FOR i := 0 TO _config.MaxControledUnits DO
    IF _controlledUnits[i] <> 0 THEN
        _status.State.AllInAuto := _status.State.AllInAuto AND _controlledUnits[i].StatusInfo.Mode = eCUMode.AutomatMode;
        _status.State.AllInManual := _status.State.AllInManual AND _controlledUnits[i].StatusInfo.Mode = eCUMode.ManualMode;
        _status.State.AllIdle := _status.State.AllIdle AND _controlledUnits[i].StatusInfo.Mode = eCUMode.NoMode;
        _status.State.AllInGrounding := _status.State.AllInGrounding AND
            (_controlledUnits[i].StatusInfo.Mode = eCUMode.GroundModeDone XOR
            _controlledUnits[i].StatusInfo.Mode = eCUMode.GroundMode);
        _status.State.AllGrounded := _status.State.AllGrounded AND _controlledUnits[i].StatusInfo.Mode = eCUMode.GroundModeDone;
        _status.State.AllInStepMode := _status.State.AllInStepMode AND _controlledUnits[i].StatusInfo.CurrentIsInStepMode;
        _status.State.AllSuspended := _status.State.AllSuspended AND _controlledUnits[i].SuspendTask.Task.Done;
		_status.State.AllRecovered := _status.State.AllRecovered AND _controlledUnits[i].RecoverTask.Task.Done;
		_status.State.AllInactiveOrManualOrGrounded := _status.State.AllInactiveOrManualOrGrounded 
											AND (_controlledUnits[i].StatusInfo.Mode = eCUMode.ManualMode 
												OR _controlledUnits[i].StatusInfo.Mode = eCUMode.NoMode 
												OR _controlledUnits[i].StatusInfo.Mode = eCUMode.GroundModeDone );
		
        _status.State.AnyInAuto := _status.State.AnyInAuto OR _controlledUnits[i].StatusInfo.Mode = eCUMode.AutomatMode;
        _status.State.AnyInManual := _status.State.AnyInManual OR _controlledUnits[i].StatusInfo.Mode = eCUMode.ManualMode;
        _status.State.AnyInStepMode := _status.State.AnyInStepMode OR _controlledUnits[i].StatusInfo.CurrentIsInStepMode;
        _status.State.AnyGrounding := _status.State.AnyGrounding OR
            (_controlledUnits[i].StatusInfo.Mode = eCUMode.GroundModeDone OR
            _controlledUnits[i].StatusInfo.Mode = eCUMode.GroundMode);

    ELSE
        EXIT;
    END_IF
END_FOR

// update states of buttons
_status.State.AnyButtonRecover := FALSE;
_status.State.AnyButtonSuspend := FALSE;
_status.State.AnyButtonGround := FALSE;
_status.State.AnyButtonAuto := FALSE;
i := 0;

FOR i := 0 TO _config.MaxControlButtons DO
    IF _controlButtons[i] <> 0 THEN
        _status.State.AnyButtonRecover := _status.State.AnyButtonRecover OR _controlButtons[i].ButtonRecover;
        _status.State.AnyButtonGround := _status.State.AnyButtonGround OR _controlButtons[i].ButtonGround;
        _status.State.AnyButtonAuto := _status.State.AnyButtonAuto OR _controlButtons[i].ButtonAuto;
        _status.State.AnyButtonSuspend := _status.State.AnyButtonSuspend OR _controlButtons[i].ButtonSuspend;
    ELSE
        EXIT;
    END_IF
END_FOR

// update states of keys
_status.State.AllKeysNormal := TRUE;
_status.State.AnyKeyService := FALSE;
i := 0;

FOR i := 0 TO _config.MaxKeyNormalService DO
    IF _controlKeyNormalService[i] <> 0 THEN
        _status.State.AllKeysNormal := _status.State.AllKeysNormal AND _controlKeyNormalService[i].KeyInNormal;
        _status.State.AnyKeyService := _status.State.AnyKeyService OR _controlKeyNormalService[i].KeyInService;
    ELSE
        EXIT;
    END_IF
END_FOR

// update states of keys
_status.State.AllKeysAuto := TRUE;
_status.State.AnyKeyManual := FALSE;
_status.State.AnyKeyStep := FALSE;
i := 0;

FOR i := 0 TO _config.MaxKeyMode DO
    IF _controlKeyMode[i] <> 0 THEN
        _status.State.AllKeysAuto := _status.State.AllKeysAuto AND _controlKeyMode[i].KeyInAuto;
        _status.State.AnyKeyManual := _status.State.AnyKeyManual OR _controlKeyMode[i].KeyInManual;
        _status.State.AnyKeyStep := _status.State.AnyKeyStep OR _controlKeyMode[i].KeyInStep;
    ELSE
        EXIT;
    END_IF
END_FOR
END_METHOD

METHOD KeyAuto 
VAR
	cu : UINT;
END_VAR
IF _keyAutoTask.Execute() THEN
	_status.ActionDescription:= '<#Automatic mode is not possibe to set(All keys must be in NORMAL and AUTO!)#>';
	IF 	 _status.State.AllKeysNormal  AND _status.State.AllKeysAuto THEN
		
//			_status.ActionDescription:= '<#Automatic mode is set(Step mode is disabled)!#>';
//			FOR cu := 0 TO _config.MaxControledUnits DO
//				IF _controlledUnits[cu] <> 0 THEN
//					IF _controlledUnits[cu].StatusInfo.Mode=eCUMode.AutomatMode THEN
//						_controlledUnits[cu].AutomatTask.ModeController.Mode:=eSequencerMode.CyclicMode;
//					ELSIF _controlledUnits[cu].StatusInfo.Mode=eCUMode.GroundMode THEN
//						_controlledUnits[cu].GroundTask.ModeController.Mode:=eSequencerMode.CyclicMode;
//					END_IF
//				ELSE
//					EXIT;
//				END_IF
//			END_FOR
	
		ELSE
			_status.ActionDescription:= '<#Cyclic mode is not allowed while any control key is in Service mode!#> <#Setting step mode!#>';
			FOR cu := 0 TO _config.MaxControledUnits DO
				IF _controlledUnits[cu] <> 0 THEN
						IF _controlledUnits[cu].StatusInfo.Mode=eCUMode.AutomatMode THEN
							_controlledUnits[cu].AutomatTask.ModeController.Mode:=eSequencerMode.StepMode;
						ELSIF _controlledUnits[cu].StatusInfo.Mode=eCUMode.GroundMode THEN
							_controlledUnits[cu].GroundTask.ModeController.Mode:=eSequencerMode.StepMode;
						END_IF
				ELSE
					EXIT;
				END_IF
			END_FOR	
		END_IF;
	
	


	IF  _status.State.AllInAuto THEN
		_keyAutoTask.DoneWhen(TRUE);
	END_IF;
	
	IF _status.ActionDescription<>'' THEN
		THIS^._keyAutoTask.Messenger.Notify(_status.ActionDescription);
	END_IF;	
END_IF
END_METHOD

METHOD KeyManual 
VAR
	cu : UINT;
END_VAR

IF _keyManualTask.Execute() THEN
	_status.ActionDescription:= '<#Manual mode is not possibe to set(At least one SERVICE and one MANUAL keys must be in position!)#>';
	
	IF _keyManualTask.Progress =0 THEN
		IF _status.State.AnyKeyManual AND _status.State.AnyKeyService THEN
			IF NOT _status.State.AllInManual THEN
				_keyManualTask.Progress := _keyManualTask.Progress + 1;// all to manual
			ELSE
				_keyManualTask.Progress := _keyManualTask.Progress + 2;
			END_IF
		END_IF;
	
	END_IF

	IF _keyManualTask.Progress =1 THEN
		
		_status.ActionDescription:='<#Manual mode is starting#>';
		
		FOR cu := 0 TO _config.MaxControledUnits DO
			IF _controlledUnits[cu] <> 0 THEN
				IF  _controlledUnits[cu].StatusInfo.Mode<> eCUMode.ManualMode THEN
					_controlledUnits[cu].ManualTask.Invoke();
				END_IF			
			ELSE
				EXIT;
			END_IF
		END_FOR

		IF _status.State.AllInManual THEN
			_keyManualTask.Progress := _keyManualTask.Progress + 1;
		END_IF
		
	END_IF
	
	
	IF _keyManualTask.Progress =2 THEN
		
		_status.ActionDescription:='<#Clear step mode#>';
		
		FOR cu := 0 TO _config.MaxControledUnits DO
			IF _controlledUnits[cu] <> 0 THEN
				_controlledUnits[cu].AutomatTask.ModeController.Mode := eSequencerMode.CyclicMode;
				_controlledUnits[cu].GroundTask.ModeController.Mode := eSequencerMode.CyclicMode;		
			ELSE
				EXIT;
			END_IF
		END_FOR

		IF _status.State.AllInManual THEN
			_keyManualTask.Progress := _keyManualTask.Progress + 1;
		END_IF
		
	END_IF

	IF _keyManualTask.Progress =3 THEN
		_keyManualTask.DoneWhen(TRUE);	
	END_IF

	IF _status.ActionDescription<>'' THEN
		THIS^._keyManualTask.Messenger.Notify(_status.ActionDescription);
	END_IF;
END_IF;
END_METHOD

METHOD KeyService
VAR
	cu : UINT;
END_VAR
IF _keyServiceTask.Execute() THEN
	
	IF 	_status.State.AnyKeyManual  AND _status.State.AnyKeyService  THEN
		_status.ActionDescription:='<#Manual mode is starting due service key combination (Manual / Service)#>';
		
		FOR cu := 0 TO _config.MaxControledUnits DO
			IF _controlledUnits[cu] <> 0 THEN
				IF  _controlledUnits[cu].StatusInfo.Mode<> eCUMode.ManualMode THEN
					_controlledUnits[cu].ManualTask.Invoke();
				END_IF			
			ELSE
				EXIT;
			END_IF
		END_FOR
	ELSE
		_status.ActionDescription:='<#Step mode is required because Service key position is set!#>';
		FOR cu := 0 TO _config.MaxControledUnits DO
			IF _controlledUnits[cu] <> 0 THEN
					IF _controlledUnits[cu].StatusInfo.Mode=eCUMode.AutomatMode THEN
						_controlledUnits[cu].AutomatTask.ModeController.Mode:=eSequencerMode.StepMode;
					ELSIF _controlledUnits[cu].StatusInfo.Mode=eCUMode.GroundMode THEN
						_controlledUnits[cu].GroundTask.ModeController.Mode:=eSequencerMode.StepMode;
					END_IF
			ELSE
				EXIT;
			END_IF
		END_FOR
	END_IF;
	


	IF  _status.State.AllInStepMode OR _status.State.AllInManual THEN
		_keyServiceTask.DoneWhen(TRUE);
	END_IF;
	
	IF _status.ActionDescription<>'' THEN
		THIS^._keyServiceTask.Messenger.Notify(_status.ActionDescription);
	END_IF;	
END_IF
END_METHOD

METHOD KeyStep 
VAR
	cu : UINT;
END_VAR

IF _keyStepTask.Execute() THEN
		
	_status.ActionDescription:='<#Step mode is required but mode key is not in required position!#>';

	IF _status.State.AnyKeyStep THEN
		FOR cu := 0 TO _config.MaxControledUnits DO
			IF _controlledUnits[cu] <> 0 THEN
				IF _controlledUnits[cu].StatusInfo.Mode=eCUMode.AutomatMode THEN
					_controlledUnits[cu].AutomatTask.ModeController.Mode:=eSequencerMode.StepMode;
				ELSIF _controlledUnits[cu].StatusInfo.Mode=eCUMode.GroundMode THEN
					_controlledUnits[cu].GroundTask.ModeController.Mode:=eSequencerMode.StepMode;
				END_IF
			ELSE
				EXIT;
			END_IF
		
		END_FOR
	END_IF;
	
	IF _status.State.AllInStepMode THEN
		_status.ActionDescription:='<#Step mode is set or all are inactive!#>';
		_keyStepTask.DoneWhen(TRUE);
	END_IF;
	
	IF _status.ActionDescription<>'' THEN
		THIS^._keyStepTask.Messenger.Notify(_status.ActionDescription);
	END_IF;	
END_IF;
END_METHOD

METHOD Restore :  TcoCore.ITcoRestorable
VAR
	i : UINT;
END_VAR
// clear all linked Controlled units
FOR i := 0 TO _config.MaxControledUnits DO
	_controlledUnits[i] := 0;
END_FOR

// clear all linked Control buttons
FOR i := 0 TO _config.MaxControlButtons DO
	_controlButtons[i] := 0;
END_FOR

// clear all linked service keys (N/S)
FOR i := 0 TO _config.MaxKeyNormalService DO
	_controlKeyNormalService[i] := 0;
END_FOR

// clear all linked Sequencer keys (M/S/A)
FOR i := 0 TO _config.MaxKeyMode DO
	_controlKeyMode[i] := 0;
END_FOR


THIS^.Messenger.UnPin();
END_METHOD

(*~
	<docu>
		<summary>
		    Custom service (manual, maintenance) logic.
			This method must be implemented in derived class.
		</summary>			
	</docu>	
~*)
METHOD PROTECTED  ServiceMode
END_METHOD

METHOD Signalisation
VAR_INPUT
END_VAR

AnyButtonAuto:=_blinkerSlow.IsOn  AND _autoTask.Busy;
END_METHOD

PROPERTY Status : REFERENCE TO TcoControlledZone_Status
GET
Status REF=_status;
END_GET
END_PROPERTY

END_FUNCTION_BLOCK

// ---- Abstractions/Safety/ControlVoltage/TcoControlVoltage.TcPOU
{attribute wpf [Container(Layout.Stack)]}
FUNCTION_BLOCK TcoControlVoltage EXTENDS TcoElements.TcoDi IMPLEMENTS  ITcoControlVoltage

VAR_OUTPUT
END_VAR
VAR
END_VAR

SUPER^(inoSignal:=inoSignal);
IF NOT inoSignal THEN
	Messenger.Error('<#Voltage is Off!#>');
END_IF;

PROPERTY IsOff : BOOL
GET
IsOff:=not this^._signal;
END_GET
END_PROPERTY

PROPERTY IsOn : BOOL
GET
IsOn:=this^._signal;
END_GET
END_PROPERTY

END_FUNCTION_BLOCK

// ---- Abstractions/Safety/DoorCircuit/TcoDoorCircuit.TcPOU
FUNCTION_BLOCK TcoDoorCircuit EXTENDS TcoCore.TcoComponent IMPLEMENTS ITcoDoorCircuit
VAR_INPUT
END_VAR
VAR_OUTPUT
END_VAR
VAR
	
	{attribute addProperty Name "<#Status#>"}
    {attribute clr [ReadOnly()]}
    _status : TcoDoorCircuit_Status;

	{attribute addProperty Name "<#Config#>"}
    _config : TcoDoorCircuit_Config;

	
	{attribute clr [RenderIgnore()]}
	_doors              : ARRAY [0..12] OF ITcoDoorLock;
	
	{attribute clr [RenderIgnore()]}
	_localDoorsVoltage  : ARRAY [0..4] OF ITcoControlVoltage;
	
	{attribute clr [RenderIgnore()]}
	_localVoltage  : ARRAY [0..4] OF ITcoControlVoltage;
	
	{attribute clr [RenderIgnore()]}
	_globalVoltage : ARRAY [0..4] OF ITcoControlVoltage;
	
	
	
    {attribute addProperty Name "<#Closed#>"}
    _isClosed : BOOL;
    
    {attribute addProperty Name "<#Locked#>"}
    _isLocked : BOOL;
    
    {attribute addProperty Name "<#Unlocked#>"}
    _isUnLocked : BOOL;
    
    {attribute addProperty Name "<#Global votage#>"}
    _isGlobalVoltageOk : BOOL;
    
    {attribute addProperty Name "<#Local voltage#>"}
    _isLocalVoltageOk : BOOL;
    
	 {attribute addProperty Name "<#Local Doors#>"}
    _isLocalDoorsVoltageOk : BOOL;


END_VAR

Initialize();

METHOD AddDoors : BOOL
VAR_INPUT
	inDoor : ITcoDoorLock;
END_VAR
VAR
	i : UINT;
END_VAR
AddDoors := FALSE;
FOR i := 0 TO _config.MaxDoors DO
	IF _doors[i] = inDoor THEN
		AddDoors := TRUE;
		RETURN;
	END_IF
	
	IF _doors[i] = 0 THEN
		_doors[i] := inDoor;
		AddDoors := TRUE;
		RETURN;
	END_IF
END_FOR
END_METHOD

METHOD AddGlobalVoltage : BOOL
VAR_INPUT
 	inVoltage : ITcoControlVoltage;
END_VAR
VAR
	i : UINT;
END_VAR
AddGlobalVoltage := FALSE;

IF inVoltage = 0 THEN
	RETURN;
END_IF

FOR i := 0 TO _config.MaxGlobalVoltage DO
	IF _globalVoltage[i] = inVoltage THEN
		addGlobalVoltage := TRUE;
		RETURN;
	END_IF
	
	IF 	_globalVoltage[i] = 0 THEN
		_globalVoltage[i] := inVoltage;
		addGlobalVoltage    := TRUE;
		RETURN;
	END_IF
END_FOR
END_METHOD

METHOD AddLocalDoorsVoltage : BOOL
VAR_INPUT
 	inVoltage : ITcoControlVoltage;
END_VAR
VAR
	i : UINT;
END_VAR
AddLocalDoorsVoltage := FALSE;

IF inVoltage = 0 THEN
	RETURN;
END_IF

FOR i := 0 TO _config.MaxLocalVoltage DO
	IF _localDoorsVoltage[i] = inVoltage THEN
		AddLocalDoorsVoltage := TRUE;
		RETURN;
	END_IF
	
	IF 	_localDoorsVoltage[i] = 0 THEN
		_localDoorsVoltage[i] := inVoltage;
		AddLocalDoorsVoltage    := TRUE;
		RETURN;
	END_IF
END_FOR
END_METHOD

METHOD AddLocalVoltage : BOOL
VAR_INPUT
 	inVoltage : ITcoControlVoltage;
END_VAR
VAR
	i : UINT;
END_VAR
addLocalVoltage := FALSE;

IF inVoltage = 0 THEN
	RETURN;
END_IF

FOR i := 0 TO _config.MaxLocalVoltage DO
	IF _localVoltage[i] = inVoltage THEN
		addLocalVoltage := TRUE;
		RETURN;
	END_IF
	
	IF 	_localVoltage[i] = 0 THEN
		_localVoltage[i] := inVoltage;
		addLocalVoltage    := TRUE;
		RETURN;
	END_IF
END_FOR
END_METHOD

PROPERTY Config :REFERENCE TO TcoDoorCircuit_Config
GET
Config ref=_config;
END_GET
END_PROPERTY

METHOD Initialize : BOOL
VAR
	d       : UINT;
	gv      : UINT;
	lv      : UINT;
	ldoors      : UINT;
	setOnce : BOOL;
END_VAR
// ------------------------------------------------------------- 
// 						GLOBAL VOLTAGE
// ------------------------------------------------------------- 
_isGlobalVoltageOk := FALSE;
setOnce            := FALSE;

FOR gv := 0 TO _config.MaxGlobalVoltage DO
	IF _globalVoltage[gv] <> 0 THEN
		IF NOT setOnce THEN
			_isGlobalVoltageOk := TRUE;
			setOnce := TRUE;
		END_IF
		
		IF _globalVoltage[gv].IsOff THEN
			_isGlobalVoltageOk := FALSE;
			EXIT;
		END_IF
	ELSE
		EXIT;
	END_IF
END_FOR

// ------------------------------------------------------------- 
// 						LOCAL VOLTAGE
// ------------------------------------------------------------- 
_isLocalVoltageOk := FALSE;
setOnce           := FALSE;

FOR lv := 0 TO _config.MaxLocalVoltage DO
	IF _localVoltage[lv] <> 0 THEN
		IF NOT setOnce THEN
			_isLocalVoltageOk := TRUE;
			setOnce := TRUE;
		END_IF
		
		IF _localVoltage[lv].IsOff THEN
			_isLocalVoltageOk := false;
			EXIT;
		END_IF
	ELSE
		EXIT;
	END_IF
END_FOR

// ------------------------------------------------------------- 
// 						LOCAL DOORS VOLTAGE OK
// ------------------------------------------------------------- 
_isLocalDoorsVoltageOk := FALSE;
setOnce           := FALSE;

FOR ldoors := 0 TO _config.MaxLocalDoorsVoltage DO
	IF _localDoorsVoltage[ldoors] <> 0 THEN
		IF NOT setOnce THEN
			_isLocalDoorsVoltageOk := TRUE;
			setOnce := TRUE;
		END_IF
		
		IF _localDoorsVoltage[ldoors].IsOff THEN
			_isLocalDoorsVoltageOk := FALSE;
			EXIT;
		END_IF
	ELSE
		EXIT;
	END_IF
END_FOR

// ------------------------------------------------------------- 
// 							DOORS
// ------------------------------------------------------------- 
_isClosed      := FALSE;
_isLocked      := FALSE;
_isUnLocked    := FALSE;
setOnce        := FALSE;
FOR d := 0 TO _config.MaxDoors DO
	IF _doors[d] <> 0 THEN
		IF NOT setOnce THEN
			setOnce        := TRUE;
			_isClosed      := TRUE;
			_isLocked      := TRUE;
			_isUnLocked    := TRUE;
		END_IF

		// Return TRUE only if all doors are Closed
		_isClosed   := _isClosed AND (_doors[d].IsClosed); // OR _doors[d].Deactivate);
		// Return TRUE only if all doors are Locked
		_isLocked   := _isLocked AND (_doors[d].IsLocked); //OR _doors[d].Deactivate);
		// Return TRUE only if all doors are Unlocked
		_isUnLocked := _isUnLocked AND NOT _doors[d].IsLocked;

	ELSE
		EXIT;
	END_IF
END_FOR
END_METHOD

{attribute 'monitoring' := 'variable'}
PROPERTY IsClosed : BOOL
GET
VAR
	d : UINT;
	setOnce : BOOL;
END_VAR
IsClosed := _isClosed ;
END_GET
END_PROPERTY

{attribute 'monitoring' := 'variable'}
PROPERTY IsGlobalVoltageOk : BOOL
GET
VAR
	gv : UINT;
END_VAR
IsGlobalVoltageOk := _isGlobalVoltageOk;
END_GET
END_PROPERTY

{attribute 'monitoring' := 'variable'}
PROPERTY IsLocalDoorsVoltageOk : BOOL
GET
VAR
	lv : UINT;
END_VAR
IsLocalDoorsVoltageOk := _isLocalDoorsVoltageOk;
END_GET
END_PROPERTY

{attribute 'monitoring' := 'variable'}
PROPERTY IsLocalVoltageOk : BOOL
GET
VAR
	lv : UINT;
END_VAR
IsLocalVoltageOk := _isLocalVoltageOk;
END_GET
END_PROPERTY

{attribute 'monitoring' := 'variable'}
PROPERTY IsLocked : BOOL
GET
VAR
	d : UINT;
	setOnce : BOOL;
END_VAR
IsLocked := _isLocked ;
END_GET
END_PROPERTY

{attribute 'monitoring' := 'variable'}
PROPERTY IsUnLocked : BOOL
GET
VAR
	d : UINT;
	setOnce : BOOL;
END_VAR
IsUnLocked := _isUnLocked;
END_GET
END_PROPERTY

METHOD Lock : BOOL
VAR_INPUT
END_VAR
VAR
	d : UINT;
END_VAR
Lock := FALSE;

IF NOT IsClosed THEN
	// we can't lock doors which are not closed
	RETURN;
END_IF

FOR d := 0 TO _config.MaxDoors DO
	IF _doors[d] <> 0 THEN
			_doors[d].Lock();
	ELSE
		EXIT;
	END_IF
END_FOR

Lock := THIS^.IsLocked;
END_METHOD

METHOD RemoveAllDoors
VAR
	i : UINT;
END_VAR
FOR i := 0 TO _config.MaxDoors DO
	_doors[i] := 0;
END_FOR
END_METHOD

METHOD RemoveDoors : BOOL
VAR_INPUT
	inDoorLock : ITcoDoorLock;
END_VAR
VAR
	i : UINT;
END_VAR
RemoveDoors := FALSE;

FOR i := 0 TO _config.MaxDoors DO 
	IF _doors[i] = inDoorLock THEN
		_doors[i] := 0;
		RemoveDoors :=  TRUE;
		RETURN;
	END_IF
END_FOR
END_METHOD

(*~
	<docu>
		<summary>
			Restores this instance to the Ready state. Can be called explicitly or from within one of the restore mechanisms.	
		</summary>			
	</docu>	
~*)
METHOD  Restore : ITcoRestorable

VAR
	i : UINT;
END_VAR
RemoveAllDoors();

FOR i := 0 TO _config.MaxGlobalVoltage DO
	_globalVoltage[i] := 0;
END_FOR

FOR i := 0 TO _config.MaxLocalVoltage DO
	_localVoltage[i] := 0;
END_FOR
FOR i := 0 TO _config.MaxLocalDoorsVoltage DO
	_localDoorsVoltage[i] := 0;
END_FOR
END_METHOD

(*~
	<docu>
		<summary>
		    Custom service (manual, maintenance) logic.
			This method must be implemented in derived class.
		</summary>			
	</docu>	
~*)
METHOD PROTECTED  ServiceMode
END_METHOD

PROPERTY Status : REFERENCE TO TcoDoorCircuit_Status
GET
Status REF=_status;
END_GET
END_PROPERTY

METHOD UnLock : BOOL
VAR
	d 		: UINT;
	setOnce : BOOL;
END_VAR
UnLock := FALSE;

FOR d := 0 TO _config.MaxDoors DO
	IF _doors[d] <> 0 THEN
		_doors[d].Unlock();
	ELSE
		exit;
	END_IF
END_FOR


FOR d := 0 TO _config.MaxDoors DO
	IF _doors[d] <> 0 THEN
		IF NOT setOnce THEN
			setOnce := TRUE;
			UnLock := TRUE;
		END_IF
		
		// return TRUE only if all doors are unlocked
		UnLock := Unlock AND NOT _doors[d].IsLocked;
	ELSE
		EXIT;
	END_IF
END_FOR
END_METHOD

END_FUNCTION_BLOCK

// ---- Abstractions/Safety/Doors/TcoStandardDoor.TcPOU
FUNCTION_BLOCK TcoStandardDoor EXTENDS TcoCore.TcoComponent IMPLEMENTS ITcoDoorLock
VAR_IN_OUT
    inoIsOpen : BOOL;
    inoIsLocked : BOOL;
    inoLock : BOOL;
END_VAR
VAR
    {attribute addProperty Name "<#Opened#>"}
    _isOpen : TcoElements.TcoDi(THIS^);

    {attribute addProperty Name "<#Locked#>"}
    _isLocked : TcoElements.TcoDi(THIS^);

    {attribute addProperty Name "<#Lock#>"}
    _lock : TcoElements.TcoDo(THIS^);


END_VAR

THIS^._isLocked(inoSignal :=  inoIsLocked);                    
THIS^._isOpen(inoSignal :=  inoIsOpen);                    
THIS^._lock(inoSignal   :=  inoLock);

PROPERTY IsClosed : BOOL
GET
IsClosed := THIS^._isOpen.IsFalse;
END_GET
END_PROPERTY

PROPERTY IsLocked : BOOL
GET
IsLocked := THIS^._isOpen.IsFalse and THIS^._isLocked.IsTrue ;
END_GET
END_PROPERTY

PROPERTY IsOpen : BOOL
GET
IsOpen := THIS^._isOpen.IsTrue;
END_GET
END_PROPERTY

METHOD Lock : BOOL
VAR_INPUT
END_VAR
Lock := FALSE;

THIS^._lock.Set();

IF	THIS^._isOpen.IsFalse THEN 
		
	IF THIS^._isLocked.IsTrue THEN 
		Lock := TRUE;
	END_IF
END_IF
END_METHOD

(*~
	<docu>
		<summary>
			Restores this instance to the Ready state. Can be called explicitly or from within one of the restore mechanisms.	
		</summary>			
	</docu>	
~*)
METHOD  Restore : ITcoRestorable
Unlock();
END_METHOD

(*~
	<docu>
		<summary>
		    Custom service (manual, maintenance) logic.
			This method must be implemented in derived class.
		</summary>			
	</docu>	
~*)
METHOD PROTECTED  ServiceMode
END_METHOD

METHOD UnLock : BOOL
VAR_INPUT
END_VAR

UnLock := FALSE;

THIS^._lock.Reset();
		
IF THIS^._isLocked.IsFalse THEN 
	UnLock := TRUE;
END_IF
END_METHOD

END_FUNCTION_BLOCK

// ---- Abstractions/Safety/Doors/TcoBasicDoor.TcPOU
FUNCTION_BLOCK TcoBasicDoor EXTENDS TcoCore.TcoComponent IMPLEMENTS ITcoDoorLock
VAR_IN_OUT
    inoIsClosed : BOOL;
    inoLock : BOOL;
END_VAR
VAR
    {attribute addProperty Name "<#Closed#>"}
    _isClosed : TcoElements.TcoDi(THIS^);

    {attribute addProperty Name "<#Lock#>"}
    _lock : TcoElements.TcoDo(THIS^);


END_VAR

                
THIS^._isClosed(inoSignal :=  inoIsClosed);                    
THIS^._lock(inoSignal   :=  inoLock);

PROPERTY IsClosed : BOOL
GET
IsClosed := THIS^._isClosed.IsTrue;
END_GET
END_PROPERTY

PROPERTY IsLocked : BOOL
GET
IsLocked := THIS^._isClosed.IsTrue and THIS^._lock.IsTrue ;
END_GET
END_PROPERTY

PROPERTY IsOpen : BOOL
GET
IsOpen := THIS^._isClosed.IsFalse;
END_GET
END_PROPERTY

METHOD Lock : BOOL
VAR_INPUT
END_VAR
Lock := FALSE;

THIS^._lock.Set();

IF	THIS^._isClosed.IsTrue THEN 
		Lock := TRUE;
END_IF
END_METHOD

(*~
	<docu>
		<summary>
			Restores this instance to the Ready state. Can be called explicitly or from within one of the restore mechanisms.	
		</summary>			
	</docu>	
~*)
METHOD  Restore : ITcoRestorable
UnLock();
END_METHOD

(*~
	<docu>
		<summary>
		    Custom service (manual, maintenance) logic.
			This method must be implemented in derived class.
		</summary>			
	</docu>	
~*)
METHOD PROTECTED  ServiceMode
END_METHOD

METHOD UnLock : BOOL
VAR_INPUT
END_VAR

UnLock := FALSE;

THIS^._lock.Reset();
		

UnLock := TRUE;
END_METHOD

END_FUNCTION_BLOCK

// ---- Abstractions/Safety/Estop/TcoEmergencyStop.TcPOU
{attribute wpf [Container(Layout.Stack)]}
FUNCTION_BLOCK TcoEmergencyStop EXTENDS TcoElements.TcoDi
VAR_OUTPUT
END_VAR
VAR
END_VAR

SUPER^(inoSignal:=inoSignal);
IF inoSignal THEN
	Messenger.Error('<#Emergency stop active#>').Pin();
END_IF;

END_FUNCTION_BLOCK

// ---- Abstractions/Safety/KeyMode/TcoKeyMode.TcPOU
{attribute wpf [Container(Layout.Stack)]}
FUNCTION_BLOCK TcoKeyMode EXTENDS TcoCore.TcoComponent IMPLEMENTS ITcoKeyMode
VAR_IN_OUT
	{attribute clr [RenderIgnore()]}
	inoKeyState1               : BOOL;
	
	{attribute clr [RenderIgnore()]}
	inoKeyState2               : BOOL;
END_VAR
VAR	
	
	{attribute addProperty Name "<#Status#>"}
    {attribute clr [ReadOnly()]}
    _status : TcoKeyMode_Status;

	{attribute addProperty Name "<#Config#>"}
    _config : TcoKeyMode_Config;
	{attribute addProperty Name "<#KeyState1#>"}
	KeyState1                : TcoElements.TcoDi(THIS^);
	
	{attribute addProperty Name "<#KeyState2#>"}
	KeyState2                : TcoElements.TcoDi(THIS^);
	
	//----------------- KEY STATES--------------
	{attribute addProperty Name "<#Manual#>"}
	IsKeyInManual            : BOOL; 
	
	{attribute addProperty Name "<#Automatic#>"}
	IsKeyInAuto              : BOOL; 
	
	{attribute addProperty Name "<#Step mode#>"}
	IsKeyInStep              : BOOL; 
	
	
	{attribute clr [RenderIgnore()]}
	_timer:ton;
END_VAR

KeyState1(inoSignal:= inoKeyState1);
KeyState2(inoSignal:= inoKeyState2);
_timer(IN:=(NOT KeyState1._signal   AND  KeyState2._signal) XOR (KeyState1._signal   AND  NOT KeyState2._signal),PT:=_config.SwitKeyStanilisiation);
THIS^.IsKeyInAuto   := KeyState1._signal       AND  KeyState2._signal;
THIS^.IsKeyInStep   := (NOT KeyState1._signal   AND  KeyState2._signal) XOR (KeyState1._signal   AND  NOT KeyState2._signal) AND _timer.Q;
THIS^.IsKeyInManual := NOT KeyState1._signal   AND  NOT KeyState2._signal;
//todo  timer

PROPERTY Config :REFERENCE TO TcoKeyMode_Config
GET
Config ref=_config;
END_GET
END_PROPERTY

PROPERTY KeyInAuto : BOOL
GET
KeyInAuto := IsKeyInAuto;
END_GET
END_PROPERTY

PROPERTY KeyInManual : BOOL
GET
KeyInManual := IsKeyInManual;
END_GET
END_PROPERTY

PROPERTY KeyInStep : BOOL
GET
KeyInStep := IsKeyInStep;
END_GET
END_PROPERTY

(*~
	<docu>
		<summary>
			Restores this instance to the Ready state. Can be called explicitly or from within one of the restore mechanisms.	
		</summary>			
	</docu>	
~*)
METHOD  Restore : ITcoRestorable
END_METHOD

(*~
	<docu>
		<summary>
		    Custom service (manual, maintenance) logic.
			This method must be implemented in derived class.
		</summary>			
	</docu>	
~*)
METHOD PROTECTED  ServiceMode
END_METHOD

PROPERTY Status : REFERENCE TO TcoKeyMode_Status
GET
Status REF=_status;
END_GET
END_PROPERTY

END_FUNCTION_BLOCK

// ---- Abstractions/Safety/KeyNormalService/TcoKeyNormalService.TcPOU
{attribute wpf [Container(Layout.Stack)]}
FUNCTION_BLOCK TcoKeyNormalService EXTENDS TcoElements.TcoDi IMPLEMENTS ITcoKeyNormalSevice

VAR

	
	{attribute addProperty Name "<#Key state#> - <#Service#>"}
	_isKeyInService           : BOOL; 

	{attribute addProperty Name "<#Key state#> - <#Normal#>"}
	_isKeyInNormal            : BOOL; 
END_VAR

SUPER^(inoSignal:= inoSignal);


THIS^._isKeyInNormal :=NOT THIS^._signal ;
THIS^._isKeyInService := NOT THIS^._isKeyInNormal;

PROPERTY KeyInNormal : BOOL
GET
KeyInNormal := _isKeyInNormal;
END_GET
END_PROPERTY

PROPERTY KeyInService : BOOL
GET
KeyInService := _isKeyInService;
END_GET
END_PROPERTY

END_FUNCTION_BLOCK
